KUKA KRL program: lacopia.src, lacopia.dat

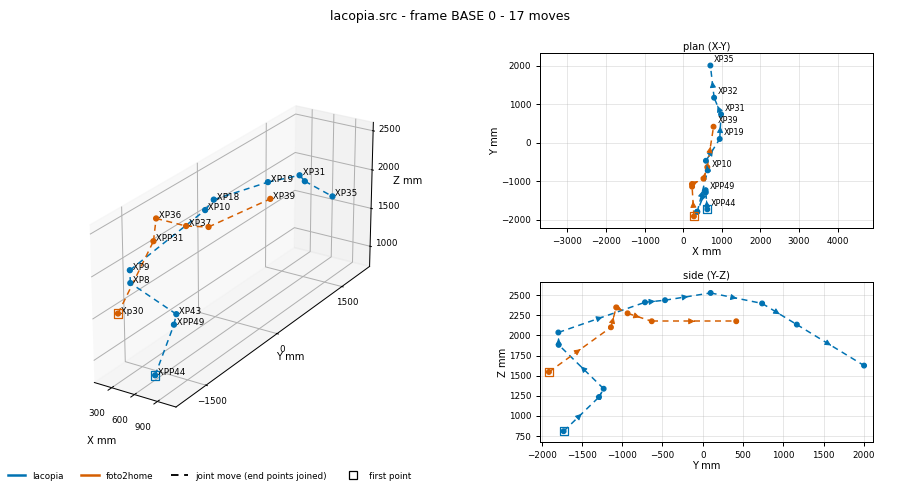
[picture p0: tool path of lacopia.src in frame BASE 0, 17 of 28 moves have a stored position in this frame; points joined in program order, loops and branches not executed]
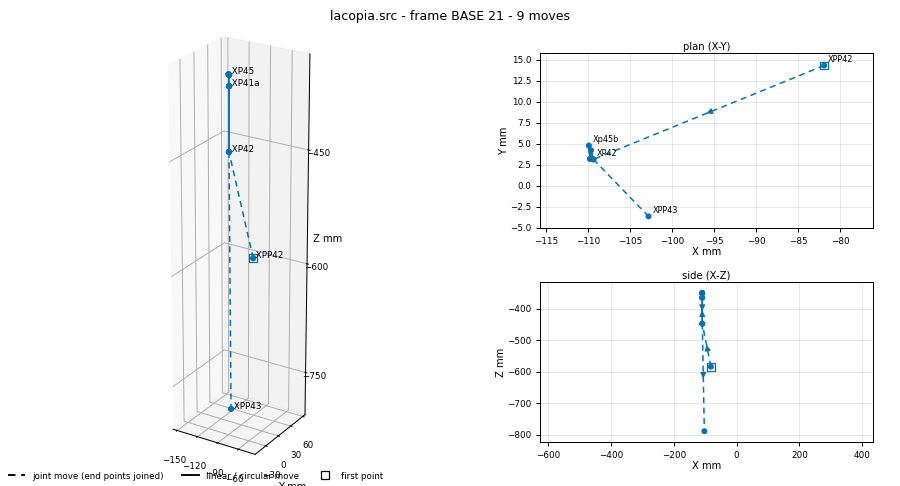
[picture p1: tool path of lacopia.src in frame BASE 21, 9 of 28 moves have a stored position in this frame; points joined in program order, loops and branches not executed]
--- lacopia.src ---
&ACCESS RVP1
&PARAM EDITMASK = *
DEF lacopia( )

;================================================
; MODELO   :
; IE GRUPO : FIP
; ESTACION : ST101
; ROBOT    : 101R1
; FUNCION  : PICK IP
;================================================

;FOLD INI
  ;FOLD BASISTECH INI
    GLOBAL INTERRUPT DECL 3 WHEN $STOPMESS==TRUE DO IR_STOPM ( )
    INTERRUPT ON 3
    BAS (#INITMOV,0 )
  ;ENDFOLD (BASISTECH INI)
;FOLD SPOTTECH INI
;USERSPOT(#INIT)
;ENDFOLD (SPOTTECH INI)
;FOLD GRIPPERTECH INI
USER_GRP(0,DUMMY,DUMMY,GDEFAULT)
INTERRUPT DECL 20 WHEN $FLAG[20]==FALSE DO GRPS(#MON_ERR,20)
;ENDFOLD (GRIPPERTECH INI)
  ;FOLD USER INI
    ;Make your modifications here
;INTERRUPT DECL 13 WHEN $IN[133]==true do stopsrch()
I_DATOS_NOK=FALSE
  ;ENDFOLD (USER INI)
;ENDFOLD (INI)


;inicializacion griper
;fold grp init
;ENTRAR_DEDOS()
;CERRAR_DEDOS()
;ENTRAR_RODILLO()
;ABRIR_CILINDRO_IP()
;CLAMPAR_GONDOLA()
;endfold
;WAIT POSITION


;ENTRADA

;===========================================================
;POSICION FOTO 1 (selccionar esta linea para repetir foto 1)
;===========================================================
;FOLD OUT 38 'PETICION A DISPOSITIVO 6' State=FALSE ;%{PE}%R 5.6.13,%MKUKATPBASIS,%COUT,%VOUTX,%P 2:38, 3:PETICION A DISPOSITIVO 6, 5:FALSE, 6:
$OUT[38]=FALSE
;ENDFOLD
;FOLD PTP PP46 Vel=100 % PDAT41 Tool[14]:camara Base[19]:carrusel bien;%{PE}%R 5.6.13,%MKUKATPBASIS,%CMOVE,%VPTP,%P 1:PTP, 2:PP46, 3:, 5:100, 7:PDAT41
$BWDSTART=FALSE
PDAT_ACT=PPDAT41
FDAT_ACT=FPP46
BAS(#PTP_PARAMS,100)
PTP XPP46
;ENDFOLD
;wait sec 1

;CHEQUEO SEÑALES RESETEADAS
MAFELEC_TECH (#CHECK_RESET, 0,0,0)

;PIDE FOTO 1
;FOLD FORDTECH.Tool_Rel 2 ;%{PE}%MKUKATPUSER
TOOL_REL (2)
;ENDFOLD

;PIDE RESULTADO FOTO
MAFELEC_TECH (#type, 0,0,0)

;EVALUA RESULTADO FOTO
switch I_TYPE_INFO
case 2
o_type_req=FALSE
;FOLD FORDTECH.Tool_Req 2 ;%{PE}%MKUKATPUSER
TOOL_REQ (2)
;ENDFOLD
foto2home()
goto home
endswitch

base_data[21]=base_data[19]
;APLICA CORRECCIONES A BASE
MAFELEC_TECH (#GET_CORR, 21,0,0)

tool_data[16]=tool_data[14]
;APLICA CORRECCION ANGULO A TOOL
MAFELEC_TECH (#GET_CORR_TOOL,16 ,0,0)

;REGISTRA CORRECCIONES
MAFELEC_TECH (#REG1, 5,0,0)

;FINALIZA PROCESO CORRECCIONES
o_type_req=false
wait for i_type_info==0
;FOLD FORDTECH.Tool_Req 2 ;%{PE}%MKUKATPUSER
TOOL_REQ (2)
;ENDFOLD

;POSICION FOTO 2


xpp45=xpp46
;FOLD PTP PP45 Vel=100 % PDAT37 Tool[16]:camara_corregida Base[21]:carrusel_corregido;%{PE}%R 5.6.13,%MKUKATPBASIS,%CMOVE,%VPTP,%P 1:PTP, 2:PP45, 3:, 5:100, 7:PDAT37
$BWDSTART=FALSE
PDAT_ACT=PPDAT37
FDAT_ACT=FPP45
BAS(#PTP_PARAMS,100)
PTP XPP45
;ENDFOLD


;wait sec 1

;PIDE FOTO 2
;FOLD FORDTECH.Tool_Rel 6 ;%{PE}%MKUKATPUSER
TOOL_REL (6)
;ENDFOLD

;PIDE RESULTADO FOTO
MAFELEC_TECH (#type, 0,0,0)

;EVALUA RESULTADO FOTO
switch I_TYPE_INFO
case 1 ;foto ok
o_type_req=false
wait for i_type_info==0
case 2 ;foto no ok
o_type_req=FALSE
;FOLD FORDTECH.Tool_Req 6 ;%{PE}%MKUKATPUSER
TOOL_REQ (6)
;ENDFOLD
foto2home()
goto home
endswitch
;FINALIZA PRODCESO FOTO 2
;FOLD FORDTECH.Tool_Req 6 ;%{PE}%MKUKATPUSER
TOOL_REQ (6)
;ENDFOLD

if not i_dry then

;FOLD CHEQUEO LIMITE SEGUNDO OFFSET
;WAIT FOR OHCbase_OFFSETz>-200
;WAIT FOR OHCbase_OFFSETz<200
;WAIT FOR OHCbase_OFFSETx>-200
;WAIT FOR OHCbase_OFFSETx<200
;WAIT FOR OHCtool_OFFSETb>-0.200
;WAIT FOR OHCtool_OFFSETb<0.370
;ENDFOLD
;APLICAMOS OFFSET
;FOLD OFFSET CORR
;BASE_DATA[7].Z=OHCbase_CORR.Z+OHCbase_OFFSETz
;BASE_DATA[7].X=OHCbase_CORR.X+OHCbase_OFFSETx
;TOOL_DATA[5].B=OHCtool_CORR.B+OHCtool_OFFSETb
;ENDFOLD

;FOLD WAIT FOR ( IN 72 '201S167B agarre IP abierto izq' ) CONT;%{PE}%R 5.6.13,%MKUKATPBASIS,%CEXT_WAIT_FOR,%VEXT_WAIT_FOR,%P 2:, 4:, 5:$IN, 6:72, 7:201S167B agarre IP abierto izq, 9:CONTINUE
CONTINUE
WAIT FOR  ( $IN[72] )
;ENDFOLD
;FOLD WAIT FOR ( IN 104 '201S168B agarre IP abierto drch' ) CONT;%{PE}%R 5.6.13,%MKUKATPBASIS,%CEXT_WAIT_FOR,%VEXT_WAIT_FOR,%P 2:, 4:, 5:$IN, 6:104, 7:201S168B agarre IP abierto drch, 9:CONTINUE
CONTINUE
WAIT FOR  ( $IN[104] )
;ENDFOLD

;FOLD WAIT FOR ( IN 98 '201S162B dedos atras drch' ) CONT;%{PE}%R 5.6.13,%MKUKATPBASIS,%CEXT_WAIT_FOR,%VEXT_WAIT_FOR,%P 2:, 4:, 5:$IN, 6:98, 7:201S162B dedos atras drch, 9:CONTINUE
CONTINUE
WAIT FOR  ( $IN[98] )
;ENDFOLD
;FOLD WAIT FOR ( IN 66 '201S161B dedos dentro izq' ) CONT;%{PE}%R 5.6.13,%MKUKATPBASIS,%CEXT_WAIT_FOR,%VEXT_WAIT_FOR,%P 2:, 4:, 5:$IN, 6:66, 7:201S161B dedos dentro izq, 9:CONTINUE
CONTINUE
WAIT FOR  ( $IN[66] )
;ENDFOLD

;FOLD WAIT FOR ( IN 102 '201S166B rodilllo dentro drch' ) CONT;%{PE}%R 5.6.13,%MKUKATPBASIS,%CEXT_WAIT_FOR,%VEXT_WAIT_FOR,%P 2:, 4:, 5:$IN, 6:102, 7:201S166B rodilllo dentro drch, 9:CONTINUE
CONTINUE
WAIT FOR  ( $IN[102] )
;ENDFOLD
;FOLD WAIT FOR ( IN 70 '201S165B rodillos izq dentro' ) CONT;%{PE}%R 5.6.13,%MKUKATPBASIS,%CEXT_WAIT_FOR,%VEXT_WAIT_FOR,%P 2:, 4:, 5:$IN, 6:70, 7:201S165B rodillos izq dentro, 9:CONTINUE
CONTINUE
WAIT FOR  ( $IN[70] )
;ENDFOLD

;FOLD WAIT FOR ( IN 100 '201S164B dedo cerrado drch' ) CONT;%{PE}%R 5.6.13,%MKUKATPBASIS,%CEXT_WAIT_FOR,%VEXT_WAIT_FOR,%P 2:, 4:, 5:$IN, 6:100, 7:201S164B dedo cerrado drch, 9:CONTINUE
CONTINUE
WAIT FOR  ( $IN[100] )
;ENDFOLD
;FOLD WAIT FOR ( IN 68 '201S163B dedos CERRADO izq' ) CONT;%{PE}%R 5.6.13,%MKUKATPBASIS,%CEXT_WAIT_FOR,%VEXT_WAIT_FOR,%P 2:, 4:, 5:$IN, 6:68, 7:201S163B dedos CERRADO izq, 9:CONTINUE
CONTINUE
WAIT FOR  ( $IN[68] )
;ENDFOLD

;FOLD WAIT FOR ( IN 105 '201S1610B nilon cerrado drch' ) CONT;%{PE}%R 5.6.13,%MKUKATPBASIS,%CEXT_WAIT_FOR,%VEXT_WAIT_FOR,%P 2:, 4:, 5:$IN, 6:105, 7:201S1610B nilon cerrado drch, 9:CONTINUE
CONTINUE
WAIT FOR  ( $IN[105] )
;ENDFOLD
;FOLD WAIT FOR ( IN 73 '201S169B nilon cerrado izq' ) CONT;%{PE}%R 5.6.13,%MKUKATPBASIS,%CEXT_WAIT_FOR,%VEXT_WAIT_FOR,%P 2:, 4:, 5:$IN, 6:73, 7:201S169B nilon cerrado izq, 9:CONTINUE
CONTINUE
WAIT FOR  ( $IN[73] )
;ENDFOLD

;PUNTO ENTRADA A COGIDA
;INTERRUPT ON 13
;wait for false
;goto alejandro
;FOLD PTP PP42 CONT Vel=100 % PDAT35 Tool[16]:camara_corregida Base[21]:carrusel_corregido;%{PE}%R 5.6.13,%MKUKATPBASIS,%CMOVE,%VPTP,%P 1:PTP, 2:PP42, 3:C_PTP, 5:100, 7:PDAT35
$BWDSTART=FALSE
PDAT_ACT=PPDAT35
FDAT_ACT=FPP42
BAS(#PTP_PARAMS,100)
PTP XPP42 C_PTP
;ENDFOLD

;PICK POSITION
;FOLD PTP P42 CONT Vel=100 % PDAT58 Tool[16]:camara_corregida Base[21]:carrusel_corregido;%{PE}%R 5.6.13,%MKUKATPBASIS,%CMOVE,%VPTP,%P 1:PTP, 2:P42, 3:C_PTP, 5:100, 7:PDAT58
$BWDSTART=FALSE
PDAT_ACT=PPDAT58
FDAT_ACT=FP42
BAS(#PTP_PARAMS,100)
PTP XP42 C_PTP
;ENDFOLD
;FOLD LIN P41a CONT Vel=2 m/s L Tool[16]:camara_corregida Base[21]:carrusel_corregido;%{PE}%R 5.6.13,%MKUKATPBASIS,%CMOVE,%VLIN,%P 1:LIN, 2:P41a, 3:C_DIS, 5:2, 7:L
$BWDSTART=FALSE
LDAT_ACT=LL
FDAT_ACT=FP41a
BAS(#CP_PARAMS,2)
LIN XP41a C_DIS
;ENDFOLD
;FOLD LIN P45 Vel=2 m/s L Tool[16]:camara_corregida Base[21]:carrusel_corregido;%{PE}%R 5.6.13,%MKUKATPBASIS,%CMOVE,%VLIN,%P 1:LIN, 2:P45, 3:, 5:2, 7:L
$BWDSTART=FALSE
LDAT_ACT=LL
FDAT_ACT=FP45
BAS(#CP_PARAMS,2)
LIN XP45
;ENDFOLD



;FOLD LIN p45b Vel=2 m/s L Tool[16]:camara_corregida Base[21]:carrusel_corregido;%{PE}%R 5.6.13,%MKUKATPBASIS,%CMOVE,%VLIN,%P 1:LIN, 2:p45b, 3:, 5:2, 7:L
$BWDSTART=FALSE
LDAT_ACT=LL
FDAT_ACT=Fp45b
BAS(#CP_PARAMS,2)
LIN Xp45b
;ENDFOLD

;FOLD LIN p45r Vel=2 m/s L Tool[16]:camara_corregida Base[21]:carrusel_corregido;%{PE}%R 5.6.13,%MKUKATPBASIS,%CMOVE,%VLIN,%P 1:LIN, 2:p45r, 3:, 5:2, 7:L
$BWDSTART=FALSE
LDAT_ACT=LL
FDAT_ACT=Fp45r
BAS(#CP_PARAMS,2)
LIN Xp45r
;ENDFOLD


if false then
endif

;Aumenta sensibilidad TORQ MON


SET_TQ_VALUES (30,30,30,30,30,30)

;cerrar_CILINDRO_IP_r()

CERRAR_CILINDRO_IP_rod()
;WAIT SEC 0.5
;SACAR_RODILLO()
;WAIT SEC 0.5
DESCLAMPAR_GONDOLA()
;WAIT SEC 0.5
CLAMPAR_GONDOLA()
;ENTRAR_RODILLO()

;espera detector IP 201S176 a 1
WAIT FOR ( $IN[109] )

;FOLD LIN p42a Vel=0.04 m/s L Tool[16]:camara_corregida Base[21]:carrusel_corregido;%{PE}%R 5.6.13,%MKUKATPBASIS,%CMOVE,%VLIN,%P 1:LIN, 2:p42a, 3:, 5:0.04, 7:L
$BWDSTART=FALSE
LDAT_ACT=LL
FDAT_ACT=Fp42a
BAS(#CP_PARAMS,0.04)
LIN Xp42a
;ENDFOLD
;FOLD LIN P42 CONT Vel=2 m/s L2 Tool[16]:camara_corregida Base[21]:carrusel_corregido;%{PE}%R 5.6.13,%MKUKATPBASIS,%CMOVE,%VLIN,%P 1:LIN, 2:P42, 3:C_DIS, 5:2, 7:L2
$BWDSTART=FALSE
LDAT_ACT=LL2
FDAT_ACT=FP42
BAS(#CP_PARAMS,2)
LIN XP42 C_DIS
;ENDFOLD
;FOLD PTP PP43 CONT Vel=100 % PDAT63 Tool[16]:camara_corregida Base[21]:carrusel_corregido;%{PE}%R 5.6.13,%MKUKATPBASIS,%CMOVE,%VPTP,%P 1:PTP, 2:PP43, 3:C_PTP, 5:100, 7:PDAT63
$BWDSTART=FALSE
PDAT_ACT=PPDAT63
FDAT_ACT=FPP43
BAS(#PTP_PARAMS,100)
PTP XPP43 C_PTP
;ENDFOLD


;espera detector IP 201S176 a 1
WAIT FOR ( $IN[109] )

endif

;TRAYECTORIA ALEJAMIENTO BALANCINA

;FOLD OUT 107 'freno garra ip' State=FALSE ;%{PE}%R 5.6.13,%MKUKATPBASIS,%COUT,%VOUTX,%P 2:107, 3:freno garra ip, 5:FALSE, 6:
$OUT[107]=FALSE
;ENDFOLD

;CHEQUEO IP COGIDO
;FOLD FORDTECH.Tool_Rel 1 ;%{PE}%MKUKATPUSER
TOOL_REL (1)
;ENDFOLD
;FOLD FORDTECH.Tool_Req 1 ;%{PE}%MKUKATPUSER
TOOL_REQ (1)
;ENDFOLD


;FOLD SYN OUT 101 'meter rodillo' State=TRUE at START Delay=0 ms;%{PE}%R 5.6.13,%MKUKATPBASIS,%COUT,%VSYNOUT,%P 2:101, 3:meter rodillo, 5:TRUE, 7:0, 9:0, 12:0
TRIGGER WHEN DISTANCE=0 DELAY=0 DO $OUT[101]=TRUE
;ENDFOLD
;FOLD SYN OUT 102 'sacar rodilllo' State=FALSE at START Delay=0 ms;%{PE}%R 5.6.13,%MKUKATPBASIS,%COUT,%VSYNOUT,%P 2:102, 3:sacar rodilllo, 5:FALSE, 7:0, 9:0, 12:0
TRIGGER WHEN DISTANCE=0 DELAY=0 DO $OUT[102]=FALSE
;ENDFOLD
;FOLD SYN OUT 97 'dedos fuera' State=TRUE at START Delay=0 ms;%{PE}%R 5.6.13,%MKUKATPBASIS,%COUT,%VSYNOUT,%P 2:97, 3:dedos fuera, 5:TRUE, 7:0, 9:0, 12:0
TRIGGER WHEN DISTANCE=0 DELAY=0 DO $OUT[97]=TRUE
;ENDFOLD
;FOLD SYN OUT 98 'dedos dentro' State=FALSE at START Delay=0 ms;%{PE}%R 5.6.13,%MKUKATPBASIS,%COUT,%VSYNOUT,%P 2:98, 3:dedos dentro, 5:FALSE, 7:0, 9:0, 12:0
TRIGGER WHEN DISTANCE=0 DELAY=0 DO $OUT[98]=FALSE
;ENDFOLD

;Deja TORQMON en valores nominales
SET_TQ_VALUES ( )

;FOLD PTP PP44 CONT Vel=100 % PDAT36 Tool[16]:camara_corregida Base[21]:carrusel_corregido;%{PE}%R 5.6.13,%MKUKATPBASIS,%CMOVE,%VPTP,%P 1:PTP, 2:PP44, 3:C_PTP, 5:100, 7:PDAT36
$BWDSTART=FALSE
PDAT_ACT=PPDAT36
FDAT_ACT=FPP44
BAS(#PTP_PARAMS,100)
PTP XPP44 C_PTP
;ENDFOLD
;FOLD PTP PP49 CONT Vel=100 % PDAT42 Tool[14]:camara Base[0];%{PE}%R 5.6.13,%MKUKATPBASIS,%CMOVE,%VPTP,%P 1:PTP, 2:PP49, 3:C_PTP, 5:100, 7:PDAT42
$BWDSTART=FALSE
PDAT_ACT=PPDAT42
FDAT_ACT=FPP49
BAS(#PTP_PARAMS,100)
PTP XPP49 C_PTP
;ENDFOLD
;FOLD PTP P43 CONT Vel=100 % PDAT60 Tool[14]:camara Base[0];%{PE}%R 5.6.13,%MKUKATPBASIS,%CMOVE,%VPTP,%P 1:PTP, 2:P43, 3:C_PTP, 5:100, 7:PDAT60
$BWDSTART=FALSE
PDAT_ACT=PPDAT60
FDAT_ACT=FP43
BAS(#PTP_PARAMS,100)
PTP XP43 C_PTP
;ENDFOLD

;libera area 1
;FOLD FORDTECH.Area_Rel 1 ;%{PE}%MKUKATPUSER
;AREA_REL (1)
;ENDFOLD
;FOLD SYN OUT 17 'LIBERACION AREA 1 carrus' State=TRUE at START Delay=0 ms;%{PE}%R 5.6.13,%MKUKATPBASIS,%COUT,%VSYNOUT,%P 2:17, 3:LIBERACION AREA 1 carrus, 5:TRUE, 7:0, 9:0, 12:0
TRIGGER WHEN DISTANCE=0 DELAY=0 DO $OUT[17]=TRUE
;ENDFOLD
;FOLD FORDTECH.Job_Rdy 1 , 1 ;%{PE}%MKUKATPUSER
JOB_READY (1,1)
;ENDFOLD
$TIMER_STOP[2]=TRUE

;FOLD PTP P8 CONT Vel=100 % PDAT43 Tool[13] Base[0];%{PE}%R 5.6.13,%MKUKATPBASIS,%CMOVE,%VPTP,%P 1:PTP, 2:P8, 3:C_PTP, 5:100, 7:PDAT43
$BWDSTART=FALSE
PDAT_ACT=PPDAT43
FDAT_ACT=FP8
BAS(#PTP_PARAMS,100)
PTP XP8 C_PTP
;ENDFOLD

;FOLD PTP P9 CONT Vel=100 % PDAT44 Tool[13] Base[0];%{PE}%R 5.6.13,%MKUKATPBASIS,%CMOVE,%VPTP,%P 1:PTP, 2:P9, 3:C_PTP, 5:100, 7:PDAT44
$BWDSTART=FALSE
PDAT_ACT=PPDAT44
FDAT_ACT=FP9
BAS(#PTP_PARAMS,100)
PTP XP9 C_PTP
;ENDFOLD


;giro
;FOLD PTP P10 CONT Vel=90 % M Tool[13] Base[0];%{PE}%R 5.6.13,%MKUKATPBASIS,%CMOVE,%VPTP,%P 1:PTP, 2:P10, 3:C_PTP, 5:90, 7:M
$BWDSTART=FALSE
PDAT_ACT=PM
FDAT_ACT=FP10
BAS(#PTP_PARAMS,90)
PTP XP10 C_PTP
;ENDFOLD

;FOLD PTP P18 CONT Vel=90 % M Tool[13] Base[0];%{PE}%R 5.6.13,%MKUKATPBASIS,%CMOVE,%VPTP,%P 1:PTP, 2:P18, 3:C_PTP, 5:90, 7:M
$BWDSTART=FALSE
PDAT_ACT=PM
FDAT_ACT=FP18
BAS(#PTP_PARAMS,90)
PTP XP18 C_PTP
;ENDFOLD
;FOLD PTP P19 CONT Vel=90 % M Tool[13] Base[0];%{PE}%R 5.6.13,%MKUKATPBASIS,%CMOVE,%VPTP,%P 1:PTP, 2:P19, 3:C_PTP, 5:90, 7:M
$BWDSTART=FALSE
PDAT_ACT=PM
FDAT_ACT=FP19
BAS(#PTP_PARAMS,90)
PTP XP19 C_PTP
;ENDFOLD
;FOLD PTP P31 CONT Vel=90 % M Tool[13] Base[0];%{PE}%R 5.6.13,%MKUKATPBASIS,%CMOVE,%VPTP,%P 1:PTP, 2:P31, 3:C_PTP, 5:90, 7:M
$BWDSTART=FALSE
PDAT_ACT=PM
FDAT_ACT=FP31
BAS(#PTP_PARAMS,90)
PTP XP31 C_PTP
;ENDFOLD
;FOLD PTP P32 Vel=90 % M Tool[13] Base[0];%{PE}%R 5.6.13,%MKUKATPBASIS,%CMOVE,%VPTP,%P 1:PTP, 2:P32, 3:, 5:90, 7:M
$BWDSTART=FALSE
PDAT_ACT=PM
FDAT_ACT=FP32
BAS(#PTP_PARAMS,90)
PTP XP32
;ENDFOLD

sacar_DEDOS()
ENTRAR_RODILLO()

;wait area ems
alejandro:

;TRAYECTORIA SALIDA AREA
;FOLD PTP P35 Vel=70 % PDAT52 Tool[13] Base[0];%{PE}%R 5.6.13,%MKUKATPBASIS,%CMOVE,%VPTP,%P 1:PTP, 2:P35, 3:, 5:70, 7:PDAT52
$BWDSTART=FALSE
PDAT_ACT=PPDAT52
FDAT_ACT=FP35
BAS(#PTP_PARAMS,70)
PTP XP35
;ENDFOLD

;TRABAJO FINALIZADO Y AREA LIBRE

home:
END
def stopsrch()
brake
resume
end
def foto2home()

;FOLD FORDTECH.Tool_Req 2 ;%{PE}%MKUKATPUSER
TOOL_REQ (2)
;ENDFOLD
SACAR_DEDOS ( )
;FOLD PTP p30 CONT Vel=15 % PDAT24 Tool[0] Base[0];%{PE}%R 5.6.13,%MKUKATPBASIS,%CMOVE,%VPTP,%P 1:PTP, 2:p30, 3:C_PTP, 5:15, 7:PDAT24
$BWDSTART=FALSE
PDAT_ACT=PPDAT24
FDAT_ACT=Fp30
BAS(#PTP_PARAMS,15)
PTP Xp30 C_PTP
;ENDFOLD
;FOLD PTP PP31 Vel=15 % PDAT26 Tool[1]:weld Base[0];%{PE}%R 5.6.13,%MKUKATPBASIS,%CMOVE,%VPTP,%P 1:PTP, 2:PP31, 3:, 5:15, 7:PDAT26
$BWDSTART=FALSE
PDAT_ACT=PPDAT26
FDAT_ACT=FPP31
BAS(#PTP_PARAMS,15)
PTP XPP31
;ENDFOLD
;FOLD PTP P36 Vel=100 % PDAT53 Tool[1]:weld Base[0];%{PE}%R 5.6.13,%MKUKATPBASIS,%CMOVE,%VPTP,%P 1:PTP, 2:P36, 3:, 5:100, 7:PDAT53
$BWDSTART=FALSE
PDAT_ACT=PPDAT53
FDAT_ACT=FP36
BAS(#PTP_PARAMS,100)
PTP XP36
;ENDFOLD
;FOLD PTP P37 Vel=100 % PDAT54 Tool[1]:weld Base[0];%{PE}%R 5.6.13,%MKUKATPBASIS,%CMOVE,%VPTP,%P 1:PTP, 2:P37, 3:, 5:100, 7:PDAT54
$BWDSTART=FALSE
PDAT_ACT=PPDAT54
FDAT_ACT=FP37
BAS(#PTP_PARAMS,100)
PTP XP37
;ENDFOLD
;FOLD PTP P38 Vel=100 % PDAT55 Tool[1]:weld Base[0];%{PE}%R 5.6.13,%MKUKATPBASIS,%CMOVE,%VPTP,%P 1:PTP, 2:P38, 3:, 5:100, 7:PDAT55
$BWDSTART=FALSE
PDAT_ACT=PPDAT55
FDAT_ACT=FP38
BAS(#PTP_PARAMS,100)
PTP XP38
;ENDFOLD
;FOLD PTP P39 Vel=100 % PDAT56 Tool[1]:weld Base[0];%{PE}%R 5.6.13,%MKUKATPBASIS,%CMOVE,%VPTP,%P 1:PTP, 2:P39, 3:, 5:100, 7:PDAT56
$BWDSTART=FALSE
PDAT_ACT=PPDAT56
FDAT_ACT=FP39
BAS(#PTP_PARAMS,100)
PTP XP39
;ENDFOLD
;FOLD FORDTECH.Area_Rel 1 ;%{PE}%MKUKATPUSER
AREA_REL (1)
;ENDFOLD
I_DATOS_NOK=TRUE
end

--- lacopia.dat ---
&ACCESS RVP1
&PARAM EDITMASK = *
DEFDAT lacopia
;FOLD EXTERNAL DECLARATIONS;%{PE}%MKUKATPBASIS,%CEXT,%VCOMMON,%P
;FOLD GRIPPERTECH EXT
EXT  H50 (INT  :IN,INT  :IN,INT  :IN,GRP_TYP  :IN )
;ENDFOLD (GRIPPERTECH EXT)
;FOLD SPOTTECH EXT
EXT  USERSPOT (S_COMMAND  :IN,SPOT_TYPE  :IN )
;ENDFOLD (SPOTTECH EXT)
;FOLD BASISTECH EXT;%{PE}%MKUKATPBASIS,%CEXT,%VEXT,%P
EXT  BAS (BAS_COMMAND  :IN,REAL  :IN )
DECL INT SUCCESS
;ENDFOLD (BASISTECH EXT)
;FOLD USER EXT;%{E}%MKUKATPUSER,%CEXT,%VEXT,%P
;Make here your modifications

;ENDFOLD (USER EXT)
;ENDFOLD (EXTERNAL DECLARATIONS)
DECL BASIS_SUGG_T LAST_BASIS={POINT1[] "p46_16                  ",POINT2[] "p46_16                  ",CP_PARAMS[] "L                       ",PTP_PARAMS[] "PDAT62                  ",CONT[] "                        ",CP_VEL[] "2                       ",PTP_VEL[] "100                     ",SYNC_PARAMS[] "SYNCDAT                 ",SPL_NAME[] "S0                      "}
DECL E6POS XP1={X 2006.93005,Y -531.951721,Z 1725.58203,A -144.850006,B 73.9743805,C -130.710297,S 2,T 2,E1 0.0,E2 0.0,E3 0.0,E4 0.0,E5 0.0,E6 0.0}
DECL FDAT FP1={TOOL_NO 0,BASE_NO 0,IPO_FRAME #BASE,POINT2[] " ",TQ_STATE FALSE}
DECL PDAT PPDAT1={VEL 100.0,ACC 100.0,APO_DIST 100.0}
DECL E6POS XP2={X 1854.495,Y -933.601074,Z 1725.61401,A -156.722397,B 73.9748764,C -130.705994,S 2,T 2,E1 0.0,E2 0.0,E3 0.0,E4 0.0,E5 0.0,E6 0.0}
DECL FDAT FP2={TOOL_NO 0,BASE_NO 0,IPO_FRAME #BASE,POINT2[] " ",TQ_STATE FALSE}
DECL PDAT PPDAT2={VEL 100.0,ACC 100.0,APO_DIST 100.0}
DECL E6POS XP3={X 38.229351,Y 70.7744675,Z 37.3208084,A -0.214638695,B -1.16773498,C -0.59399718,S 2,T 42,E1 0.0,E2 0.0,E3 0.0,E4 0.0,E5 0.0,E6 0.0}
DECL FDAT FP3={TOOL_NO 3,BASE_NO 7,IPO_FRAME #BASE,POINT2[] " ",TQ_STATE FALSE}
DECL PDAT PPDAT3={VEL 100.0,ACC 100.0,APO_DIST 100.0}
DECL E6POS XP4={X 36.8946686,Y 70.8676605,Z -260.229095,A -0.293648213,B -0.9510777,C -0.591230273,S 2,T 42,E1 0.0,E2 0.0,E3 0.0,E4 0.0,E5 0.0,E6 0.0}
DECL FDAT FP4={TOOL_NO 3,BASE_NO 7,IPO_FRAME #BASE,POINT2[] " ",TQ_STATE FALSE}
DECL PDAT PPDAT4={VEL 100.0,ACC 100.0,APO_DIST 100.0}
DECL E6POS XP5={X 1562.28796,Y 893.286072,Z 1286.09705,A -15.2613897,B 0.657769501,C -90.4761124,S 2,T 3,E1 0.0,E2 0.0,E3 0.0,E4 0.0,E5 0.0,E6 0.0}
DECL FDAT FP5={TOOL_NO 3,BASE_NO 0,IPO_FRAME #BASE,POINT2[] " ",TQ_STATE FALSE}
DECL PDAT PPDAT5={VEL 100.0,ACC 100.0,APO_DIST 100.0}
DECL LDAT LCPDAT5={VEL 2.0,ACC 100.0,APO_DIST 100.0,APO_FAC 50.0,ORI_TYP #VAR,CIRC_TYP #BASE,JERK_FAC 50.0,EXAX_IGN 0}
DECL E6POS XP6={X 32.6845093,Y 70.5147781,Z -293.346405,A -0.294387609,B -0.952187896,C -0.591742516,S 2,T 42,E1 0.0,E2 0.0,E3 0.0,E4 0.0,E5 0.0,E6 0.0}
DECL FDAT FP6={TOOL_NO 3,BASE_NO 7,IPO_FRAME #BASE,POINT2[] " ",TQ_STATE FALSE}
DECL PDAT PPDAT6={VEL 100.0,ACC 100.0,APO_DIST 100.0,APO_MODE #CPTP}
DECL E6POS XP7={X 3027.01807,Y -822.159912,Z 1081.90601,A -166.794601,B -2.90207911,C -92.1657867,S 2,T 42,E1 0.0,E2 0.0,E3 0.0,E4 0.0,E5 0.0,E6 0.0}
DECL FDAT FP7={TOOL_NO 3,BASE_NO 0,IPO_FRAME #BASE,POINT2[] " ",TQ_STATE FALSE}
DECL PDAT PPDAT7={VEL 100.0,ACC 100.0,APO_DIST 100.0,APO_MODE #CPTP}
DECL PDAT PPDAT8={VEL 100.0,ACC 100.0,APO_DIST 100.0}
DECL E6POS XP11={X 41.1222,Y 69.2957764,Z -104.396698,A -0.214701205,B -1.16772699,C -0.593899012,S 2,T 42,E1 0.0,E2 0.0,E3 0.0,E4 0.0,E5 0.0,E6 0.0}
DECL FDAT FP11={TOOL_NO 3,BASE_NO 7,IPO_FRAME #BASE,POINT2[] " ",TQ_STATE FALSE}
DECL LDAT LCPDAT1={VEL 2.0,ACC 100.0,APO_DIST 100.0,APO_FAC 50.0,ORI_TYP #VAR,CIRC_TYP #BASE,JERK_FAC 50.0,EXAX_IGN 0}
DECL LDAT LCPDAT2={VEL 2.0,ACC 100.0,APO_DIST 100.0,APO_FAC 50.0,ORI_TYP #VAR,CIRC_TYP #BASE,JERK_FAC 50.0,EXAX_IGN 0}
DECL E6POS XP12={X -3.72842503,Y -101.429901,Z -620.324585,A 1.50974405,B -7.10329819,C -0.0856683701,S 2,T 42,E1 0.0,E2 0.0,E3 0.0,E4 0.0,E5 0.0,E6 0.0}
DECL FDAT FP12={TOOL_NO 3,BASE_NO 7,IPO_FRAME #BASE,POINT2[] " ",TQ_STATE FALSE}
DECL PDAT PPDAT9={VEL 100.0,ACC 100.0,APO_DIST 100.0}
DECL E6POS XP13={X 3048.49609,Y -726.61377,Z 1252.05298,A -165.1026,B 0.675549388,C -90.7842712,S 2,T 42,E1 0.0,E2 0.0,E3 0.0,E4 0.0,E5 0.0,E6 0.0}
DECL FDAT FP13={TOOL_NO 10,BASE_NO 0,IPO_FRAME #BASE,POINT2[] " ",TQ_STATE FALSE}
DECL PDAT PPDAT10={VEL 100.0,ACC 100.0,APO_DIST 100.0}
DECL E6POS XP14={X 26.6935005,Y 202.252304,Z -440.791107,A -0.295880914,B -0.950786889,C -0.591688991,S 2,T 42,E1 0.0,E2 0.0,E3 0.0,E4 0.0,E5 0.0,E6 0.0}
DECL FDAT FP14={TOOL_NO 3,BASE_NO 5,IPO_FRAME #BASE,POINT2[] " ",TQ_STATE FALSE}
DECL PDAT PPDAT11={VEL 100.0,ACC 100.0,APO_DIST 100.0}
DECL PDAT PPDAT12={VEL 100.0,ACC 100.0,APO_DIST 100.0}
DECL E6POS XP15={X 32.5107689,Y 164.632507,Z -741.100403,A -0.294008106,B -0.952496827,C -0.591114283,S 2,T 42,E1 0.0,E2 0.0,E3 0.0,E4 0.0,E5 0.0,E6 0.0}
DECL FDAT FP15={TOOL_NO 3,BASE_NO 5,IPO_FRAME #BASE,POINT2[] " ",TQ_STATE FALSE}
DECL E6POS XP16={X 64.192421,Y 45.188961,Z -975.683777,A -2.90687799,B -12.7255402,C -0.869226217,S 2,T 42,E1 0.0,E2 0.0,E3 0.0,E4 0.0,E5 0.0,E6 0.0}
DECL FDAT FP16={TOOL_NO 3,BASE_NO 5,IPO_FRAME #BASE,POINT2[] " ",TQ_STATE FALSE}
DECL PDAT PPDAT13={VEL 100.0,ACC 100.0,APO_DIST 100.0,APO_MODE #CPTP}
DECL E6POS XP17={X 45.9537392,Y 202.007004,Z -417.451599,A -0.295843989,B -0.95071882,C -0.591725171,S 2,T 42,E1 0.0,E2 0.0,E3 0.0,E4 0.0,E5 0.0,E6 0.0}
DECL FDAT FP17={TOOL_NO 3,BASE_NO 5,IPO_FRAME #BASE,POINT2[] " ",TQ_STATE FALSE}
DECL PDAT PPDAT14={VEL 100.0,ACC 100.0,APO_DIST 100.0,APO_MODE #CPTP}
DECL PDAT PPDAT15={VEL 100.0,ACC 100.0,APO_DIST 100.0}
DECL E6POS XP_={X 3061.59497,Y -131.053894,Z 1146.73999,A -154.179092,B -2.21626902,C -91.8224716,S 2,T 43,E1 0.0,E2 0.0,E3 0.0,E4 0.0,E5 0.0,E6 0.0}
DECL FDAT Fp_={TOOL_NO 3,BASE_NO 0,IPO_FRAME #BASE,POINT2[] " ",TQ_STATE FALSE}
DECL PDAT PPDAT16={VEL 100.0,ACC 100.0,APO_DIST 100.0}
DECL E6POS XP20={X 41.1222,Y 69.2957764,Z -104.396698,A -0.214701205,B -1.16772699,C -0.593899012,S 2,T 42,E1 0.0,E2 0.0,E3 0.0,E4 0.0,E5 0.0,E6 0.0}
DECL FDAT Fp20={TOOL_NO 3,BASE_NO 7,IPO_FRAME #BASE,POINT2[] " ",TQ_STATE FALSE}
DECL LDAT LCPDAT3={VEL 2.0,ACC 100.0,APO_DIST 100.0,APO_FAC 50.0,ORI_TYP #VAR,CIRC_TYP #BASE,JERK_FAC 50.0,EXAX_IGN 0}
DECL E6POS XP21={X 1742.49902,Y 144.840897,Z -738.127808,A 6.21827412,B 75.8271179,C 4.77260399,S 2,T 10,E1 0.0,E2 0.0,E3 0.0,E4 0.0,E5 0.0,E6 0.0}
DECL FDAT Fp21={TOOL_NO 10,BASE_NO 6,IPO_FRAME #BASE,POINT2[] " ",TQ_STATE FALSE}
DECL PDAT PPDAT17={VEL 100.0,ACC 100.0,APO_DIST 100.0,APO_MODE #CPTP}
DECL E6POS XP22={X 2993.78296,Y -282.495789,Z 1156.71399,A -162.6474,B -2.34018302,C -91.4635925,S 2,T 43,E1 0.0,E2 0.0,E3 0.0,E4 0.0,E5 0.0,E6 0.0}
DECL FDAT Fp22={TOOL_NO 3,BASE_NO 0,IPO_FRAME #BASE,POINT2[] " ",TQ_STATE FALSE}
DECL PDAT PPDAT18={VEL 100.0,ACC 100.0,APO_DIST 100.0}
;DECL E6POS XP23={X 27.6339493,Y 202.200104,Z -440.799408,A -0.293876112,B -0.951247573,C -0.591240585,S 2,T 42,E1 0.0,E2 0.0,E3 0.0,E4 0.0,E5 0.0,E6 0.0}
;copiado el xp15
DECL E6POS XP23={X 32.5107689,Y 164.632507,Z -741.100403,A -0.294008106,B -0.952496827,C -0.591114283,S 2,T 42,E1 0.0,E2 0.0,E3 0.0,E4 0.0,E5 0.0,E6 0.0}
DECL FDAT Fp23={TOOL_NO 5,BASE_NO 7,IPO_FRAME #BASE,POINT2[] " ",TQ_STATE FALSE}
DECL PDAT PPDAT19={VEL 100.0,ACC 100.0,APO_DIST 100.0}
DECL E6POS XP24={X 25.8778591,Y 72.9977722,Z 38.7192001,A -0.133837,B -1.27465403,C 0.233077407,S 2,T 42,E1 0.0,E2 0.0,E3 0.0,E4 0.0,E5 0.0,E6 0.0}
DECL FDAT Fp24={TOOL_NO 5,BASE_NO 7,IPO_FRAME #BASE,POINT2[] " ",TQ_STATE FALSE}
DECL LDAT LCPDAT4={VEL 2.0,ACC 100.0,APO_DIST 100.0,APO_FAC 50.0,ORI_TYP #VAR,CIRC_TYP #BASE,JERK_FAC 50.0,EXAX_IGN 0}
DECL E6POS XP25={X 26.7191792,Y 73.1574326,Z 44.2344818,A -0.295453101,B -1.13712204,C 0.235855207,S 2,T 42,E1 0.0,E2 0.0,E3 0.0,E4 0.0,E5 0.0,E6 0.0}
DECL FDAT Fp25={TOOL_NO 5,BASE_NO 7,IPO_FRAME #BASE,POINT2[] " ",TQ_STATE FALSE}
DECL PDAT PPDAT20={VEL 100.0,ACC 100.0,APO_DIST 100.0}
DECL LDAT LCPDAT6={VEL 2.0,ACC 100.0,APO_DIST 100.0,APO_FAC 50.0,ORI_TYP #VAR,CIRC_TYP #BASE,JERK_FAC 50.0,EXAX_IGN 0}
DECL E6POS XP26={X 35.2218513,Y 74.7988968,Z -383.483795,A -0.293857187,B -1.13707495,C 0.236622602,S 2,T 42,E1 0.0,E2 0.0,E3 0.0,E4 0.0,E5 0.0,E6 0.0}
DECL FDAT Fp26={TOOL_NO 5,BASE_NO 7,IPO_FRAME #BASE,POINT2[] " ",TQ_STATE FALSE}
DECL PDAT PPDAT21={VEL 100.0,ACC 100.0,APO_DIST 100.0}
DECL E6POS XP27={X 35.2068596,Y 66.6177063,Z -383.559998,A -0.293789595,B -1.13695598,C 0.236545101,S 2,T 42,E1 0.0,E2 0.0,E3 0.0,E4 0.0,E5 0.0,E6 0.0}
DECL FDAT Fp27={TOOL_NO 5,BASE_NO 7,IPO_FRAME #BASE,POINT2[] " ",TQ_STATE FALSE}
DECL LDAT LCPDAT7={VEL 2.0,ACC 100.0,APO_DIST 100.0,APO_FAC 50.0,ORI_TYP #VAR,CIRC_TYP #BASE,JERK_FAC 50.0,EXAX_IGN 0}
DECL E6POS XP28={X 47.9414215,Y -197.943497,Z -893.239685,A 1.98645496,B -12.0790796,C 0.142493293,S 2,T 42,E1 0.0,E2 0.0,E3 0.0,E4 0.0,E5 0.0,E6 0.0}
DECL FDAT Fp28={TOOL_NO 5,BASE_NO 7,IPO_FRAME #BASE,POINT2[] " ",TQ_STATE FALSE}
DECL PDAT PPDAT22={VEL 100.0,ACC 100.0,APO_DIST 100.0,APO_MODE #CPTP}
DECL E6POS XP29={X 1499.53003,Y 259.302887,Z -582.508423,A 2.58441901,B 55.6062889,C 1.72372401,S 2,T 10,E1 0.0,E2 0.0,E3 0.0,E4 0.0,E5 0.0,E6 0.0}
DECL FDAT Fp29={TOOL_NO 10,BASE_NO 6,IPO_FRAME #BASE,POINT2[] " ",TQ_STATE FALSE}
DECL PDAT PPDAT23={VEL 100.0,ACC 100.0,APO_DIST 100.0}
DECL E6POS XP30={X 278.475586,Y -1908.98804,Z 1545.66394,A -179.522293,B 44.2849312,C -178.149902,S 2,T 10,E1 0.0,E2 0.0,E3 0.0,E4 0.0,E5 0.0,E6 0.0}
DECL FDAT Fp30={TOOL_NO 0,BASE_NO 0,IPO_FRAME #BASE,POINT2[] " ",TQ_STATE FALSE}
DECL PDAT PPDAT24={VEL 100.0,ACC 100.0,APO_DIST 100.0,APO_MODE #CPTP}
DECL PDAT PPDAT25={VEL 100.0,ACC 100.0,APO_DIST 100.0,APO_MODE #CPTP}
DECL E6POS XPP31={X 230.806702,Y -1139.68506,Z 2100.01196,A -88.1130219,B 61.2092094,C -87.0944672,S 2,T 10,E1 0.0,E2 0.0,E3 0.0,E4 0.0,E5 0.0,E6 0.0}
DECL FDAT FPP31={TOOL_NO 1,BASE_NO 0,IPO_FRAME #BASE,POINT2[] " ",TQ_STATE FALSE}
DECL PDAT PPDAT26={VEL 100.0,ACC 100.0,APO_DIST 100.0}
DECL E6POS XPP32={X 881.059814,Y 161.003296,Z -631.478088,A 1.49337006,B 15.2436895,C 0.637633979,S 2,T 3,E1 0.0,E2 0.0,E3 0.0,E4 0.0,E5 0.0,E6 0.0}
DECL FDAT FPP32={TOOL_NO 3,BASE_NO 6,IPO_FRAME #BASE,POINT2[] " ",TQ_STATE FALSE}
DECL PDAT PPDAT27={VEL 100.0,ACC 100.0,APO_DIST 100.0}
DECL LDAT LL={VEL 2.0,ACC 30.0,APO_DIST 100.0,APO_FAC 50.0,ORI_TYP #VAR,CIRC_TYP #BASE,JERK_FAC 50.0,EXAX_IGN 0}
DECL E6POS XPP33={X 27.4540195,Y 73.2977219,Z 7.42760515,A -0.295086414,B -1.13691103,C 0.236272097,S 2,T 42,E1 0.0,E2 0.0,E3 0.0,E4 0.0,E5 0.0,E6 0.0}
DECL FDAT FPP33={TOOL_NO 5,BASE_NO 7,IPO_FRAME #BASE,POINT2[] " ",TQ_STATE FALSE}
DECL E6POS XPP34={X 27.4416504,Y 65.1367874,Z 7.35081005,A -0.295179397,B -1.13690901,C 0.236488894,S 2,T 42,E1 0.0,E2 0.0,E3 0.0,E4 0.0,E5 0.0,E6 0.0}
DECL FDAT FPP34={TOOL_NO 5,BASE_NO 7,IPO_FRAME #BASE,POINT2[] " ",TQ_STATE FALSE}
DECL E6POS XPP35={X -107.751999,Y -9.56887722,Z -929.528625,A 89.7359772,B 0.775470078,C 0.2014011,S 2,T 10,E1 0.0,E2 0.0,E3 0.0,E4 0.0,E5 0.0,E6 0.0}
DECL FDAT FPP35={TOOL_NO 14,BASE_NO 19,IPO_FRAME #BASE,POINT2[] " ",TQ_STATE FALSE}
DECL PDAT PPDAT28={VEL 100.0,ACC 100.0,APO_DIST 100.0}
DECL E6POS XPP36={X -88.4785538,Y -267.269409,Z -651.501282,A 90.0431213,B 0.673774481,C -0.288594902,S 2,T 11,E1 0.0,E2 0.0,E3 0.0,E4 0.0,E5 0.0,E6 0.0}
DECL FDAT FPP36={TOOL_NO 10,BASE_NO 21,IPO_FRAME #BASE,POINT2[] " ",TQ_STATE FALSE}
DECL PDAT PPDAT29={VEL 100.0,ACC 100.0,APO_DIST 100.0}
DECL E6POS XPP37={X 80.8797226,Y 31.2043896,Z -770.521118,A 90.0418777,B 0.673092008,C -0.289515108,S 2,T 11,E1 0.0,E2 0.0,E3 0.0,E4 0.0,E5 0.0,E6 0.0}
DECL FDAT FPP37={TOOL_NO 5,BASE_NO 19,IPO_FRAME #BASE,POINT2[] " ",TQ_STATE FALSE}
DECL PDAT PPDAT30={VEL 100.0,ACC 100.0,APO_DIST 100.0}
DECL E6POS XPP37_aux={X 80.8797226,Y 31.2043896,Z -770.521118,A 90.0418777,B 0.673092008,C -0.289515108,S 2,T 11,E1 0.0,E2 0.0,E3 0.0,E4 0.0,E5 0.0,E6 0.0}
DECL FDAT FPP37_aux={TOOL_NO 7,BASE_NO 21,IPO_FRAME #BASE,POINT2[] " ",TQ_STATE FALSE}
DECL E6POS XPP38={X 944.80127,Y -1137.30505,Z 1648.67798,A 156.109207,B 47.9735985,C 179.273895,S 2,T 10,E1 0.0,E2 0.0,E3 0.0,E4 0.0,E5 0.0,E6 0.0}
DECL FDAT FPP38={TOOL_NO 0,BASE_NO 0,IPO_FRAME #BASE,POINT2[] " ",TQ_STATE FALSE}
DECL PDAT PPDAT31={VEL 100.0,ACC 100.0,APO_DIST 100.0}
DECL E6POS XPP39={X 751.101685,Y -873.903809,Z 1527.10999,A 156.482895,B 48.551651,C 179.774704,S 2,T 10,E1 0.0,E2 0.0,E3 0.0,E4 0.0,E5 0.0,E6 0.0}
DECL FDAT FPP39={TOOL_NO 0,BASE_NO 0,IPO_FRAME #BASE,POINT2[] " ",TQ_STATE FALSE}
DECL PDAT PPDAT32={VEL 100.0,ACC 100.0,APO_DIST 100.0}
DECL E6POS XPP40={X 1166.26196,Y -574.317017,Z 1438.01501,A -172.692596,B 50.0456886,C -177.410507,S 2,T 10,E1 0.0,E2 0.0,E3 0.0,E4 0.0,E5 0.0,E6 0.0}
DECL FDAT FPP40={TOOL_NO 0,BASE_NO 0,IPO_FRAME #BASE,POINT2[] " ",TQ_STATE FALSE}
DECL PDAT PPDAT33={VEL 100.0,ACC 100.0,APO_DIST 100.0}
DECL E6POS XPP41={X -105.161003,Y 0.918125808,Z -348.360901,A 89.9843292,B 0.590195715,C -0.167510897,S 2,T 10,E1 0.0,E2 0.0,E3 0.0,E4 0.0,E5 0.0,E6 0.0}
DECL FDAT FPP41={TOOL_NO 16,BASE_NO 21,IPO_FRAME #BASE,POINT2[] " ",TQ_STATE FALSE}
DECL PDAT PPDAT34={VEL 100.0,ACC 100.0,APO_DIST 100.0}
DECL E6POS XPP42={X -81.9365463,Y 14.3172903,Z -583.822815,A 90.033783,B 0.775862515,C 0.0466330498,S 2,T 10,E1 0.0,E2 0.0,E3 0.0,E4 0.0,E5 0.0,E6 0.0}
DECL FDAT FPP42={TOOL_NO 16,BASE_NO 21,IPO_FRAME #BASE,POINT2[] " ",TQ_STATE FALSE}
DECL PDAT PPDAT35={VEL 100.0,ACC 100.0,APO_DIST 100.0,APO_MODE #CPTP}
DECL E6POS XPP43={X -102.829697,Y -3.62723708,Z -789.168823,A 89.9807129,B 0.588879824,C -0.170724005,S 2,T 10,E1 0.0,E2 0.0,E3 0.0,E4 0.0,E5 0.0,E6 0.0}
DECL FDAT FPP43={TOOL_NO 16,BASE_NO 21,IPO_FRAME #BASE,POINT2[] " ",TQ_STATE FALSE}
DECL E6POS XPP44={X 624.882874,Y -1726.36499,Z 810.918579,A -142.996704,B 89.1323471,C -142.339493,S 2,T 10,E1 0.0,E2 0.0,E3 0.0,E4 0.0,E5 0.0,E6 0.0}
DECL FDAT FPP44={TOOL_NO 14,BASE_NO 0,IPO_FRAME #BASE,POINT2[] " ",TQ_STATE FALSE}
DECL PDAT PPDAT36={VEL 100.0,ACC 100.0,APO_DIST 100.0,APO_MODE #CPTP}
DECL E6POS XPP45={X -107.755898,Y -9.55412006,Z -929.54248,A 89.7358322,B 0.775858879,C 0.201302901,S 2,T 10,E1 0.0,E2 0.0,E3 0.0,E4 0.0,E5 0.0,E6 0.0}
DECL FDAT FPP45={TOOL_NO 16,BASE_NO 21,IPO_FRAME #BASE,POINT2[] " ",TQ_STATE FALSE}
DECL PDAT PPDAT37={VEL 100.0,ACC 100.0,APO_DIST 100.0}
DECL E6POS XPP46={X -107.755898,Y -9.55412006,Z -929.54248,A 89.7358322,B 0.775858879,C 0.201302901,S 2,T 10,E1 0.0,E2 0.0,E3 0.0,E4 0.0,E5 0.0,E6 0.0}
DECL FDAT FPP46={TOOL_NO 14,BASE_NO 19,IPO_FRAME #BASE,POINT2[] " ",TQ_STATE FALSE}
DECL PDAT PPDAT38={VEL 100.0,ACC 100.0,APO_DIST 100.0}
DECL E6POS XPP47={X 24.4180698,Y -4.78785896,Z -1202.16895,A 89.0462265,B 0.677900374,C -0.288725913,S 2,T 11,E1 0.0,E2 0.0,E3 0.0,E4 0.0,E5 0.0,E6 0.0}
DECL FDAT FPP47={TOOL_NO 14,BASE_NO 19,IPO_FRAME #BASE,POINT2[] " ",TQ_STATE FALSE}
DECL PDAT PPDAT39={VEL 100.0,ACC 100.0,APO_DIST 100.0}
DECL E6POS XPP48={X 504.720215,Y -1339.56104,Z 967.474121,A -177.350494,B 42.7763214,C 172.561096,S 2,T 10,E1 0.0,E2 0.0,E3 0.0,E4 0.0,E5 0.0,E6 0.0}
DECL FDAT FPP48={TOOL_NO 0,BASE_NO 0,IPO_FRAME #BASE,POINT2[] " ",TQ_STATE FALSE}
DECL PDAT PPDAT40={VEL 100.0,ACC 100.0,APO_DIST 100.0}
DECL PDAT PPDAT41={VEL 100.0,ACC 100.0,APO_DIST 100.0}
DECL E6POS XPP49={X 586.345886,Y -1287.74097,Z 1234.59399,A -90.7680588,B 82.6829071,C -90.0669479,S 2,T 10,E1 0.0,E2 0.0,E3 0.0,E4 0.0,E5 0.0,E6 0.0}
DECL FDAT FPP49={TOOL_NO 14,BASE_NO 0,IPO_FRAME #BASE,POINT2[] " ",TQ_STATE FALSE}
DECL PDAT PPDAT42={VEL 100.0,ACC 100.0,APO_DIST 100.0,APO_MODE #CPTP}
DECL PDAT PPDAT43={VEL 100.0,ACC 100.0,APO_DIST 100.0,APO_MODE #CPTP}
DECL E6POS XP8={X 364.633209,Y -1787.91199,Z 1882.00098,A -158.8311,B 69.1081772,C -155.869293,S 2,T 10,E1 0.0,E2 0.0,E3 0.0,E4 0.0,E5 0.0,E6 0.0}
DECL FDAT FP8={TOOL_NO 13,BASE_NO 0,IPO_FRAME #BASE,POINT2[] " ",TQ_STATE FALSE}
DECL PDAT PPDAT44={VEL 100.0,ACC 100.0,APO_DIST 100.0,APO_MODE #CPTP}
DECL E6POS XP9={X 364.964996,Y -1791.89001,Z 2035.68604,A -144.050598,B 66.4307404,C -139.920898,S 2,T 10,E1 0.0,E2 0.0,E3 0.0,E4 0.0,E5 0.0,E6 0.0}
DECL FDAT FP9={TOOL_NO 13,BASE_NO 0,IPO_FRAME #BASE,POINT2[] " ",TQ_STATE FALSE}
DECL PDAT PPDAT45={VEL 100.0,ACC 100.0,APO_DIST 100.0,APO_MODE #CPTP}
DECL E6POS XP10={X 635.720215,Y -717.147827,Z 2410.01807,A -168.260803,B 14.1872702,C 178.557098,S 2,T 10,E1 0.0,E2 0.0,E3 0.0,E4 0.0,E5 0.0,E6 0.0}
DECL FDAT FP10={TOOL_NO 13,BASE_NO 0,IPO_FRAME #BASE,POINT2[] " ",TQ_STATE FALSE}
DECL PDAT PPDAT46={VEL 100.0,ACC 100.0,APO_DIST 100.0,APO_MODE #CPTP}
DECL E6POS XP18={X 589.351379,Y -468.337097,Z 2436.07593,A -157.786194,B 16.6084003,C -176.289505,S 2,T 10,E1 0.0,E2 0.0,E3 0.0,E4 0.0,E5 0.0,E6 0.0}
DECL FDAT FP18={TOOL_NO 13,BASE_NO 0,IPO_FRAME #BASE,POINT2[] " ",TQ_STATE FALSE}
DECL PDAT PPDAT47={VEL 100.0,ACC 100.0,APO_DIST 100.0,APO_MODE #CPTP}
DECL E6POS XP19={X 946.800476,Y 97.3742676,Z 2526.12598,A -112.670303,B 16.4910603,C -176.548294,S 2,T 11,E1 0.0,E2 0.0,E3 0.0,E4 0.0,E5 0.0,E6 0.0}
DECL FDAT FP19={TOOL_NO 13,BASE_NO 0,IPO_FRAME #BASE,POINT2[] " ",TQ_STATE FALSE}
DECL PDAT PPDAT48={VEL 100.0,ACC 100.0,APO_DIST 100.0,APO_MODE #CPTP}
DECL E6POS XP31={X 981.520325,Y 735.968872,Z 2395.88599,A -60.3835602,B 46.7861595,C -152.051498,S 2,T 11,E1 0.0,E2 0.0,E3 0.0,E4 0.0,E5 0.0,E6 0.0}
DECL FDAT FP31={TOOL_NO 13,BASE_NO 0,IPO_FRAME #BASE,POINT2[] " ",TQ_STATE FALSE}
DECL PDAT PPDAT49={VEL 100.0,ACC 100.0,APO_DIST 100.0}
DECL E6POS XP32={X 801.582214,Y 1166.55701,Z 2133.69409,A -36.2449303,B 64.0939331,C -137.098602,S 2,T 11,E1 0.0,E2 0.0,E3 0.0,E4 0.0,E5 0.0,E6 0.0}
DECL FDAT FP32={TOOL_NO 13,BASE_NO 0,IPO_FRAME #BASE,POINT2[] " ",TQ_STATE FALSE}
DECL PDAT PPDAT50={VEL 100.0,ACC 100.0,APO_DIST 100.0}
DECL E6POS XP33={X 704.915588,Y 2000.79797,Z 1624.86499,A -13.2152596,B 44.7332916,C 178.322906,S 2,T 11,E1 0.0,E2 0.0,E3 0.0,E4 0.0,E5 0.0,E6 0.0}
DECL FDAT FP33={TOOL_NO 0,BASE_NO 0,IPO_FRAME #BASE,POINT2[] " ",TQ_STATE FALSE}
DECL E6POS XP34={X 320.607788,Y -2556.61597,Z 1133.505,A 179.833496,B 44.2316399,C -179.078995,S 2,T 10,E1 0.0,E2 0.0,E3 0.0,E4 0.0,E5 0.0,E6 0.0}
DECL FDAT FP34={TOOL_NO 0,BASE_NO 0,IPO_FRAME #BASE,POINT2[] " ",TQ_STATE FALSE}
DECL PDAT PPDAT51={VEL 100.0,ACC 100.0,APO_DIST 100.0}
DECL PDAT PPDAT52={VEL 100.0,ACC 100.0,APO_DIST 100.0}
DECL E6POS XP35={X 704.915588,Y 2000.79797,Z 1624.86499,A -13.2152596,B 44.7332916,C 178.322906,S 2,T 11,E1 0.0,E2 0.0,E3 0.0,E4 0.0,E5 0.0,E6 0.0}
DECL FDAT FP35={TOOL_NO 13,BASE_NO 0,IPO_FRAME #BASE,POINT2[] " ",TQ_STATE FALSE}
DECL E6POS XP36={X 226.764099,Y -1074.44299,Z 2347.30688,A -87.7077637,B 50.4100189,C -86.6066971,S 2,T 10,E1 0.0,E2 0.0,E3 0.0,E4 0.0,E5 0.0,E6 0.0}
DECL FDAT FP36={TOOL_NO 1,BASE_NO 0,IPO_FRAME #BASE,POINT2[] " ",TQ_STATE FALSE}
DECL PDAT PPDAT53={VEL 100.0,ACC 100.0,APO_DIST 100.0}
DECL E6POS XP37={X 526.068909,Y -932.987793,Z 2273.41699,A -69.0727921,B 61.6084595,C -94.4467697,S 2,T 10,E1 0.0,E2 0.0,E3 0.0,E4 0.0,E5 0.0,E6 0.0}
DECL FDAT FP37={TOOL_NO 1,BASE_NO 0,IPO_FRAME #BASE,POINT2[] " ",TQ_STATE FALSE}
DECL PDAT PPDAT54={VEL 100.0,ACC 100.0,APO_DIST 100.0}
DECL E6POS XP38={X 624.439392,Y -633.425476,Z 2174.77002,A -55.7007103,B 61.2513084,C -94.4497833,S 2,T 10,E1 0.0,E2 0.0,E3 0.0,E4 0.0,E5 0.0,E6 0.0}
DECL FDAT FP38={TOOL_NO 1,BASE_NO 0,IPO_FRAME #BASE,POINT2[] " ",TQ_STATE FALSE}
DECL PDAT PPDAT55={VEL 100.0,ACC 100.0,APO_DIST 100.0}
DECL E6POS XP39={X 786.753174,Y 414.935913,Z 2174.77002,A 17.5158997,B 61.2513084,C -94.4497833,S 2,T 11,E1 0.0,E2 0.0,E3 0.0,E4 0.0,E5 0.0,E6 0.0}
DECL FDAT FP39={TOOL_NO 1,BASE_NO 0,IPO_FRAME #BASE,POINT2[] " ",TQ_STATE FALSE}
DECL PDAT PPDAT56={VEL 100.0,ACC 100.0,APO_DIST 100.0}
DECL E6POS XP40={X 137.393799,Y -1879.63098,Z 1233.43799,A 154.507401,B 43.0224609,C -162.750198,S 2,T 10,E1 0.0,E2 0.0,E3 0.0,E4 0.0,E5 0.0,E6 0.0}
DECL FDAT FP40={TOOL_NO 0,BASE_NO 0,IPO_FRAME #BASE,POINT2[] " ",TQ_STATE FALSE}
DECL PDAT PPDAT57={VEL 100.0,ACC 100.0,APO_DIST 100.0}
DECL PDAT PM={VEL 100.0,ACC 75.0,APO_DIST 100.0,APO_MODE #CPTP}
DECL E6POS XP41={X -109.279503,Y 6.45388699,Z -349.479889,A 89.7366409,B 0.592110991,C -0.235046402,S 2,T 10,E1 0.0,E2 0.0,E3 0.0,E4 0.0,E5 0.0,E6 0.0}
DECL FDAT FP41={TOOL_NO 16,BASE_NO 21,IPO_FRAME #BASE,POINT2[] " ",TQ_STATE FALSE}
DECL E6POS XP42={X -109.383202,Y 3.15019703,Z -447.012085,A 89.8412628,B 0.584262371,C -0.148793101,S 2,T 10,E1 0.0,E2 0.0,E3 0.0,E4 0.0,E5 0.0,E6 0.0}
DECL FDAT FP42={TOOL_NO 16,BASE_NO 21,IPO_FRAME #BASE,POINT2[] " ",TQ_STATE FALSE}
DECL PDAT PPDAT58={VEL 100.0,ACC 100.0,APO_DIST 100.0,APO_MODE #CPTP}
DECL PDAT PPDAT59={VEL 100.0,ACC 100.0,APO_DIST 100.0}
DECL E6POS XP43={X 581.262878,Y -1230.01294,Z 1337.76501,A -88.1380386,B 76.5162735,C -87.397789,S 2,T 10,E1 0.0,E2 0.0,E3 0.0,E4 0.0,E5 0.0,E6 0.0}
DECL FDAT FP43={TOOL_NO 14,BASE_NO 0,IPO_FRAME #BASE,POINT2[] " ",TQ_STATE FALSE}
DECL PDAT PPDAT60={VEL 100.0,ACC 100.0,APO_DIST 100.0,APO_MODE #CPTP}
DECL E6POS XP44={X -109.316002,Y 7.51638794,Z -348.526703,A 89.7406006,B 0.593651414,C -0.234145805,S 2,T 10,E1 0.0,E2 0.0,E3 0.0,E4 0.0,E5 0.0,E6 0.0}
DECL FDAT FP44={TOOL_NO 16,BASE_NO 21,IPO_FRAME #BASE,POINT2[] " ",TQ_STATE FALSE}
DECL E6POS XP45={X -109.7938,Y 3.21634889,Z -349.166687,A 90.0218964,B 0.59707278,C -0.363495111,S 2,T 10,E1 0.0,E2 0.0,E3 0.0,E4 0.0,E5 0.0,E6 0.0}
DECL FDAT FP45={TOOL_NO 16,BASE_NO 21,IPO_FRAME #BASE,POINT2[] " ",TQ_STATE FALSE}
DECL E6POS XP46_3={X -81.9422531,Y 14.3149405,Z -583.80603,A 90.0340195,B 0.775730371,C 0.0464831106,S 2,T 10,E1 0.0,E2 0.0,E3 0.0,E4 0.0,E5 0.0,E6 0.0}
DECL FDAT Fp46_3={TOOL_NO 16,BASE_NO 21,IPO_FRAME #BASE,POINT2[] " ",TQ_STATE FALSE}
DECL PDAT PPDAT61={VEL 100.0,ACC 75.0,APO_DIST 100.0,APO_MODE #CPTP}
DECL E6POS XP46_6={X -109.280998,Y 6.46835709,Z -349.464386,A 89.7365494,B 0.592169285,C -0.510253429,S 2,T 10,E1 0.0,E2 0.0,E3 0.0,E4 0.0,E5 0.0,E6 0.0}
DECL FDAT Fp46_6={TOOL_NO 16,BASE_NO 21,IPO_FRAME #BASE,POINT2[] " ",TQ_STATE FALSE}
DECL PDAT PPDAT62={VEL 100.0,ACC 75.0,APO_DIST 100.0,APO_MODE #CPTP}
DECL E6POS XP46_7={X -107.938904,Y 2.851125,Z -399.012695,A 89.8768005,B 0.591036022,C -0.249589205,S 2,T 10,E1 0.0,E2 0.0,E3 0.0,E4 0.0,E5 0.0,E6 0.0}
DECL FDAT Fp46_7={TOOL_NO 16,BASE_NO 21,IPO_FRAME #BASE,POINT2[] " ",TQ_STATE FALSE}
DECL E6POS XP420={X -107.938904,Y 2.851125,Z -399.012695,A 89.8768005,B 0.591036022,C -0.249589205,S 2,T 10,E1 0.0,E2 0.0,E3 0.0,E4 0.0,E5 0.0,E6 0.0}
DECL FDAT Fp420={TOOL_NO 16,BASE_NO 21,IPO_FRAME #BASE,POINT2[] " ",TQ_STATE FALSE}
DECL E6POS XP42A={X -109.6791,Y 4.21750784,Z -364.208801,A 89.8673477,B 0.59233731,C -0.138509795,S 2,T 10,E1 0.0,E2 0.0,E3 0.0,E4 0.0,E5 0.0,E6 0.0}
DECL FDAT Fp42a={TOOL_NO 16,BASE_NO 21,IPO_FRAME #BASE,POINT2[] " ",TQ_STATE FALSE}
DECL LDAT LL2={VEL 2.0,ACC 75.0,APO_DIST 100.0,APO_FAC 50.0,ORI_TYP #VAR,CIRC_TYP #BASE,JERK_FAC 50.0,EXAX_IGN 0}
DECL E6POS Xp46_8={X -109.280998,Y 6.46835709,Z -349.464386,A 89.7365494,B 0.592169285,C -0.510253429,S 2,T 10,E1 0.0,E2 0.0,E3 0.0,E4 0.0,E5 0.0,E6 0.0}
DECL FDAT Fp46_8={TOOL_NO 16,BASE_NO 21,IPO_FRAME #BASE,POINT2[] " ",TQ_STATE FALSE}
DECL E6POS Xp46_9={X -81.9422531,Y 14.3149405,Z -583.80603,A 90.0340195,B 0.775730371,C 0.0464831106,S 2,T 10,E1 0.0,E2 0.0,E3 0.0,E4 0.0,E5 0.0,E6 0.0}
DECL FDAT Fp46_9={TOOL_NO 16,BASE_NO 21,IPO_FRAME #BASE,POINT2[] " ",TQ_STATE FALSE}
DECL E6POS XP41a={X -109.681702,Y 4.23003483,Z -364.221893,A 89.8679428,B 0.592475772,C -0.138354599,S 2,T 10,E1 0.0,E2 0.0,E3 0.0,E4 0.0,E5 0.0,E6 0.0}
DECL FDAT FP41a={TOOL_NO 16,BASE_NO 21,IPO_FRAME #BASE,POINT2[] " ",TQ_STATE FALSE}
DECL PDAT PPDAT63={VEL 100.0,ACC 100.0,APO_DIST 100.0,APO_MODE #CPTP}
DECL E6POS Xp46_10={X -109.805702,Y 4.63654184,Z -347.746613,A 89.8307571,B 0.595388174,C -0.218999207,S 2,T 10,E1 0.0,E2 0.0,E3 0.0,E4 0.0,E5 0.0,E6 0.0}
DECL FDAT Fp46_10={TOOL_NO 16,BASE_NO 21,IPO_FRAME #BASE,POINT2[] " ",TQ_STATE FALSE}
DECL PDAT PPDAT64={VEL 100.0,ACC 100.0,APO_DIST 100.0,APO_MODE #CPTP}
DECL E6POS Xp46_11={X -109.7938,Y 3.21634889,Z -349.166687,A 90.0218964,B 0.59707278,C -0.363495111,S 2,T 10,E1 0.0,E2 0.0,E3 0.0,E4 0.0,E5 0.0,E6 0.0}
DECL FDAT Fp46_11={TOOL_NO 16,BASE_NO 21,IPO_FRAME #BASE,POINT2[] " ",TQ_STATE FALSE}
DECL E6POS Xp46_12={X -109.7938,Y 3.21634889,Z -349.166687,A 90.0218964,B 0.59707278,C -0.363495111,S 2,T 10,E1 0.0,E2 0.0,E3 0.0,E4 0.0,E5 0.0,E6 0.0}
DECL FDAT Fp46_12={TOOL_NO 16,BASE_NO 21,IPO_FRAME #BASE,POINT2[] " ",TQ_STATE FALSE}
DECL E6POS Xp46_13={X -109.7938,Y 3.21634889,Z -349.166687,A 90.0218964,B 0.59707278,C -0.363495111,S 2,T 10,E1 0.0,E2 0.0,E3 0.0,E4 0.0,E5 0.0,E6 0.0}
DECL FDAT Fp46_13={TOOL_NO 16,BASE_NO 21,IPO_FRAME #BASE,POINT2[] " ",TQ_STATE FALSE}
DECL E6POS Xp45a={X -92.0735168,Y -1.04388106,Z -808.006287,A 89.8441162,B 0.854191899,C 0.144206598,S 2,T 10,E1 0.0,E2 0.0,E3 0.0,E4 0.0,E5 0.0,E6 0.0}
DECL FDAT Fp45a={TOOL_NO 16,BASE_NO 21,IPO_FRAME #BASE,POINT2[] " ",TQ_STATE FALSE}
DECL E6POS Xp46_14={X -109.925697,Y 4.79551315,Z -350.698486,A 89.8733063,B 0.599537611,C -0.228090405,S 2,T 10,E1 0.0,E2 0.0,E3 0.0,E4 0.0,E5 0.0,E6 0.0}
DECL FDAT Fp46_14={TOOL_NO 16,BASE_NO 21,IPO_FRAME #BASE,POINT2[] " ",TQ_STATE FALSE}
DECL E6POS Xp45b={X -109.925697,Y 4.79551315,Z -350.698486,A 89.8733063,B 0.599537611,C -0.228090405,S 2,T 10,E1 0.0,E2 0.0,E3 0.0,E4 0.0,E5 0.0,E6 0.0}
DECL FDAT Fp45b={TOOL_NO 16,BASE_NO 21,IPO_FRAME #BASE,POINT2[] " ",TQ_STATE FALSE}
DECL E6POS Xp46_15={X -109.9403,Y 2.7917459,Z -349.537811,A 89.975647,B 0.599607587,C -0.225769699,S 2,T 10,E1 0.0,E2 0.0,E3 0.0,E4 0.0,E5 0.0,E6 0.0}
DECL FDAT Fp46_15={TOOL_NO 16,BASE_NO 21,IPO_FRAME #BASE,POINT2[] " ",TQ_STATE FALSE}
DECL E6POS Xp46_16={X -109.7938,Y 3.21634889,Z -349.166687,A 90.0218964,B 0.59707278,C -0.363495111,S 2,T 10,E1 0.0,E2 0.0,E3 0.0,E4 0.0,E5 0.0,E6 0.0}
DECL FDAT Fp46_16={TOOL_NO 16,BASE_NO 21,IPO_FRAME #BASE,POINT2[] " ",TQ_STATE FALSE}
DECL E6POS Xp45r={X -109.7938,Y 3.21634889,Z -349.166687,A 90.0218964,B 0.59707278,C -0.363495111,S 2,T 10,E1 0.0,E2 0.0,E3 0.0,E4 0.0,E5 0.0,E6 0.0}
DECL FDAT Fp45r={TOOL_NO 16,BASE_NO 21,IPO_FRAME #BASE,POINT2[] " ",TQ_STATE FALSE}
ENDDAT
